LIN {X -326.728,Y -20.251,Z -40.000,A 0.015,B 0.000,C 180.000} C_DIS
LIN {X -326.353,Y -19.738,Z -40.000,A 0.015,B 0.000,C 180.000} C_DIS
LIN {X -324.173,Y -16.080,Z -40.000,A 0.015,B -0.000,C -180.000} C_DIS
LIN {X -324.033,Y -15.821,Z -40.000,A 0.015,B -0.000,C 180.000} C_DIS
LIN {X -323.375,Y -14.460,Z -40.000,A 0.015,B -0.000,C 180.000} C_DIS
LIN {X -323.235,Y -14.127,Z -40.000,A 0.015,B 0.000,C 180.000} C_DIS
LIN {X -321.515,Y -9.322,Z -40.000,A 0.015,B 0.000,C -180.000} C_DIS
LIN {X -321.341,Y -8.587,Z -40.000,A 0.015,B 0.000,C 180.000} C_DIS
LIN {X -320.684,Y -3.146,Z -40.000,A 0.015,B -0.000,C -180.000} C_DIS
LIN {X -320.667,Y -2.972,Z -40.000,A 0.015,B 0.000,C -180.000} C_DIS
LIN {X -320.518,Y -0.795,Z -40.000,A 0.015,B 0.000,C -180.000} C_DIS
LIN {X -320.520,Y -0.308,Z -40.000,A 0.015,B -0.000,C 180.000} C_DIS
LIN {X -320.740,Y 2.593,Z -40.000,A 0.015,B -0.000,C 180.000} C_DIS
LIN {X -320.791,Y 2.977,Z -40.000,A 0.015,B 0.000,C -180.000} C_DIS
LIN {X -321.349,Y 5.879,Z -40.000,A 0.015,B 0.000,C 180.000} C_DIS
LIN {X -321.416,Y 6.162,Z -40.000,A 0.015,B -0.000,C 180.000} C_DIS
LIN {X -321.819,Y 7.584,Z -40.000,A 0.015,B 0.000,C -180.000} C_DIS
LIN {X -321.946,Y 7.949,Z -40.000,A 0.015,B -0.000,C -180.000} C_DIS
LIN {X -324.346,Y 13.782,Z -40.000,A 0.015,B 0.000,C -180.000} C_DIS
LIN {X -324.544,Y 14.184,Z -40.000,A 0.015,B 0.000,C 180.000} C_DIS
LIN {X -342.684,Y 45.663,Z -40.000,A 0.015,B 0.000,C 180.000} C_DIS
LIN {X -342.906,Y 46.000,Z -40.000,A 0.015,B 0.000,C 180.000} C_DIS
LIN {X -344.864,Y 48.619,Z -40.000,A 0.015,B -0.000,C -180.000} C_DIS
LIN {X -344.919,Y 48.690,Z -40.000,A 0.015,B 0.000,C -180.000} C_DIS
LIN {X -347.449,Y 51.891,Z -40.000,A 0.015,B 0.000,C -180.000} C_DIS
LIN {X -347.826,Y 52.295,Z -40.000,A 0.015,B 0.000,C -180.000} C_DIS
LIN {X -350.266,Y 54.515,Z -40.000,A 0.015,B -0.000,C 180.000} C_DIS
LIN {X -350.603,Y 54.784,Z -40.000,A 0.015,B -0.000,C 180.000} C_DIS
LIN {X -352.993,Y 56.456,Z -40.000,A 0.015,B -0.000,C 180.000} C_DIS
LIN {X -353.258,Y 56.623,Z -40.000,A 0.015,B 0.000,C -180.000} C_DIS
LIN {X -354.709,Y 57.450,Z -40.000,A 0.015,B -0.000,C -180.000} C_DIS
LIN {X -355.032,Y 57.611,Z -40.000,A 0.015,B 0.000,C 180.000} C_DIS
LIN {X -360.836,Y 60.141,Z -40.000,A 0.015,B 0.000,C 180.000} C_DIS
LIN {X -361.547,Y 60.361,Z -40.000,A 0.015,B -0.000,C -180.000} C_DIS
LIN {X -365.901,Y 61.201,Z -40.000,A 0.015,B 0.000,C 180.000} C_DIS
LIN {X -366.162,Y 61.241,Z -40.000,A 0.015,B -0.000,C 180.000} C_DIS
LIN {X -368.338,Y 61.486,Z -40.000,A 0.015,B 0.000,C -180.000} C_DIS
LIN {X -368.781,Y 61.507,Z -40.000,A 0.015,B 0.000,C -180.000} C_DIS
LIN {X -373.497,Y 61.419,Z -40.000,A 0.015,B -0.000,C -180.000} C_DIS
LIN {X -374.399,Y 61.279,Z -40.000,A 0.015,B 0.000,C 180.000} C_DIS
LIN {X -383.592,Y 58.540,Z -40.000,A 0.015,B 0.000,C -180.000} C_DIS
LIN {X -383.923,Y 58.423,Z -40.000,A 0.015,B -0.000,C 180.000} C_DIS
LIN {X -384.920,Y 58.009,Z -40.000,A 0.015,B 0.000,C 180.000} C_DIS
LIN {X -385.722,Y 57.537,Z -40.000,A 0.015,B 0.000,C -180.000} C_DIS
LIN {X -393.652,Y 51.259,Z -40.000,A 0.015,B 0.000,C 180.000} C_DIS
LIN {X -394.115,Y 50.815,Z -40.000,A 0.015,B -0.000,C -180.000} C_DIS
LIN {X -395.224,Y 49.527,Z -40.000,A 0.015,B 0.000,C 180.000} C_DIS
LIN {X -395.515,Y 49.136,Z -40.000,A 0.015,B 0.000,C -180.000} C_DIS
LIN {X -397.824,Y 45.507,Z -40.000,A 0.015,B 0.000,C 180.000} C_DIS
LIN {X -397.891,Y 45.398,Z -40.000,A 0.015,B -0.000,C -180.000} C_DIS
LIN {X -401.772,Y 38.756,Z -40.000,A 0.015,B 0.000,C 180.000} C_DIS
LIN {X -401.996,Y 38.296,Z -40.000,A 0.015,B 0.000,C 180.000} C_DIS
LIN {X -402.542,Y 36.920,Z -40.000,A 0.015,B 0.000,C -180.000} C_DIS
LIN {X -402.687,Y 36.460,Z -40.000,A 0.015,B 0.000,C 180.000} C_DIS
LIN {X -403.779,Y 31.896,Z -40.000,A 0.015,B 0.000,C -180.000} C_DIS
LIN {X -403.787,Y 333.800,Z -40.000,A 0.015,B 0.000,C -180.000} C_DIS
LIN {X -403.730,Y 334.871,Z -40.000,A 0.015,B 0.000,C 180.000} C_DIS
LIN {X -403.533,Y 335.736,Z -40.000,A 0.015,B 0.000,C 180.000} C_DIS
LIN {X -403.418,Y 336.003,Z -40.000,A 0.015,B -0.000,C -180.000} C_DIS
LIN {X -403.034,Y 336.500,Z -39.830,A 0.015,B 0.000,C 180.000} C_DIS
LIN {X -402.624,Y 336.714,Z -39.365,A 0.015,B 0.000,C -180.000} C_DIS
LIN {X -402.458,Y 336.753,Z -38.730,A 0.015,B 0.000,C -180.000} C_DIS
$VEL.CP = 1.00000
LIN {X -402.458,Y 336.753,Z 11.000,A 0.015,B 0.000,C 180.000} C_DIS
$VEL.CP = 1.00000
LIN {X -176.907,Y 111.466,Z 11.000,A 0.015,B 0.000,C 180.000} C_DIS
$VEL.CP = 1.00000
LIN {X -176.907,Y 111.466,Z -28.231,A 0.015,B 0.000,C 180.000} C_DIS
$VEL.CP = 0.10000
LIN {X -176.826,Y 111.561,Z -28.780,A 0.015,B 0.000,C 180.000} C_DIS
LIN {X -176.608,Y 111.835,Z -29.221,A 0.015,B 0.000,C -180.000} C_DIS
LIN {X -176.404,Y 112.123,Z -29.421,A 0.015,B -0.000,C 180.000} C_DIS
LIN {X -176.196,Y 112.462,Z -29.500,A 0.015,B 0.000,C 180.000} C_DIS
LIN {X -176.625,Y 119.097,Z -29.746,A 0.015,B 0.000,C 180.000} C_DIS
LIN {X -182.895,Y 121.307,Z -29.992,A 0.015,B -0.000,C 180.000} C_DIS
LIN {X -187.390,Y 116.408,Z -30.238,A 0.015,B 0.000,C 180.000} C_DIS
LIN {X -184.650,Y 110.351,Z -30.484,A 0.015,B -0.000,C -180.000} C_DIS
LIN {X -178.003,Y 110.493,Z -30.730,A 0.015,B 0.000,C -180.000} C_DIS
LIN {X -175.523,Y 116.662,Z -30.975,A 0.015,B 0.000,C 180.000} C_DIS
LIN {X -180.223,Y 121.364,Z -31.221,A 0.015,B -0.000,C 180.000} C_DIS
LIN {X -186.394,Y 118.888,Z -31.467,A 0.015,B 0.000,C 180.000} C_DIS
LIN {X -186.539,Y 112.241,Z -31.713,A 0.015,B -0.000,C 180.000} C_DIS
LIN {X -180.483,Y 109.497,Z -31.959,A 0.015,B -0.000,C 180.000} C_DIS
LIN {X -175.582,Y 113.990,Z -32.205,A 0.015,B 0.000,C -180.000} C_DIS
LIN {X -177.789,Y 120.261,Z -32.451,A 0.015,B 0.000,C -180.000} C_DIS
LIN {X -184.423,Y 120.694,Z -32.697,A 0.015,B 0.000,C -180.000} C_DIS
LIN {X -187.426,Y 114.762,Z -32.943,A 0.015,B -0.000,C 180.000} C_DIS
LIN {X -183.150,Y 109.671,Z -33.189,A 0.015,B 0.000,C -180.000} C_DIS
LIN {X -176.789,Y 111.605,Z -33.434,A 0.015,B 0.000,C 180.000} C_DIS
LIN {X -176.070,Y 118.215,Z -33.680,A 0.015,B -0.000,C -180.000} C_DIS
LIN {X -181.867,Y 121.471,Z -33.926,A 0.015,B 0.000,C 180.000} C_DIS
LIN {X -187.137,Y 117.419,Z -34.172,A 0.015,B 0.000,C -180.000} C_DIS
LIN {X -185.480,Y 110.980,Z -34.418,A 0.015,B 0.000,C 180.000} C_DIS
LIN {X -178.907,Y 109.976,Z -34.664,A 0.015,B 0.000,C 180.000} C_DIS
LIN {X -175.404,Y 115.627,Z -34.910,A 0.015,B -0.000,C 180.000} C_DIS
LIN {X -179.225,Y 121.068,Z -35.156,A 0.015,B 0.000,C -180.000} C_DIS
LIN {X -185.729,Y 119.690,Z -35.402,A 0.015,B 0.000,C -180.000} C_DIS
LIN {X -187.016,Y 113.167,Z -35.648,A 0.015,B 0.000,C -180.000} C_DIS
LIN {X -181.522,Y 109.423,Z -35.893,A 0.015,B -0.000,C 180.000} C_DIS
LIN {X -175.921,Y 113.005,Z -36.139,A 0.015,B -0.000,C -180.000} C_DIS
LIN {X -177.016,Y 119.563,Z -36.385,A 0.015,B -0.000,C 180.000} C_DIS
LIN {X -183.478,Y 121.130,Z -36.631,A 0.015,B 0.000,C 180.000} C_DIS
LIN {X -187.456,Y 115.803,Z -36.877,A 0.015,B 0.000,C -180.000} C_DIS
LIN {X -184.119,Y 110.052,Z -37.123,A 0.015,B -0.000,C 180.000} C_DIS
LIN {X -177.520,Y 110.864,Z -37.369,A 0.015,B 0.000,C -180.000} C_DIS
LIN {X -175.675,Y 117.251,Z -37.615,A 0.015,B 0.000,C -180.000} C_DIS
LIN {X -180.825,Y 121.456,Z -37.861,A 0.015,B 0.000,C -180.000} C_DIS
LIN {X -186.715,Y 118.370,Z -38.107,A 0.015,B 0.000,C -180.000} C_DIS
LIN {X -186.189,Y 111.743,Z -38.352,A 0.015,B -0.000,C 180.000} C_DIS
LIN {X -179.887,Y 109.624,Z -38.598,A 0.015,B -0.000,C 180.000} C_DIS
LIN {X -175.464,Y 114.587,Z -38.844,A 0.015,B 0.000,C 180.000} C_DIS
LIN {X -178.292,Y 120.604,Z -39.090,A 0.015,B 0.000,C 180.000} C_DIS
LIN {X -184.937,Y 120.366,Z -39.336,A 0.015,B -0.000,C 180.000} C_DIS
LIN {X -187.326,Y 114.161,Z -39.582,A 0.015,B 0.000,C 180.000} C_DIS
LIN {X -182.558,Y 109.528,Z -39.828,A 0.015,B 0.000,C 180.000} C_DIS
LIN {X -176.424,Y 112.093,Z -40.074,A 0.015,B 0.000,C -180.000} C_DIS
LIN {X -176.376,Y 118.742,Z -40.320,A 0.015,B 0.000,C 180.000} C_DIS
LIN {X -182.471,Y 121.397,Z -40.566,A 0.015,B 0.000,C -180.000} C_DIS
LIN {X -187.306,Y 116.834,Z -40.811,A 0.015,B 0.000,C 180.000} C_DIS
LIN {X -185.008,Y 110.595,Z -41.057,A 0.015,B 0.000,C 180.000} C_DIS
LIN {X -178.368,Y 110.259,Z -41.303,A 0.015,B 0.000,C -180.000} C_DIS
LIN {X -175.452,Y 116.234,Z -41.549,A 0.015,B 0.000,C 180.000} C_DIS
LIN {X -179.802,Y 121.262,Z -41.795,A 0.015,B -0.000,C 180.000} C_DIS
LIN {X -186.134,Y 119.235,Z -42.041,A 0.015,B -0.000,C 180.000} C_DIS
LIN {X -186.757,Y 112.616,Z -42.287,A 0.015,B -0.000,C 180.000} C_DIS
LIN {X -180.913,Y 109.444,Z -42.533,A 0.015,B 0.000,C -180.000} C_DIS
LIN {X -175.702,Y 113.574,Z -42.779,A 0.015,B -0.000,C 180.000} C_DIS
LIN {X -177.453,Y 119.987,Z -43.025,A 0.015,B 0.000,C -180.000} C_DIS
LIN {X -184.040,Y 120.895,Z -43.270,A 0.015,B 0.000,C 180.000} C_DIS
LIN {X -187.461,Y 115.194,Z -43.516,A 0.015,B 0.000,C 180.000} C_DIS
LIN {X -183.560,Y 109.809,Z -43.762,A 0.015,B -0.000,C 180.000} C_DIS
LIN {X -177.077,Y 111.282,Z -44.008,A 0.015,B 0.000,C -180.000} C_DIS
LIN {X -175.886,Y 117.823,Z -44.254,A 0.015,B -0.000,C 180.000} C_DIS
LIN {X -181.434,Y 121.487,Z -44.500,A 0.015,B -0.000,C -180.000} C_DIS
LIN {X -214.171,Y 121.487,Z -44.500,A 0.015,B -0.000,C -180.000} C_DIS
CIRC {X -216.093,Y 120.378,Z -44.500,A 0.015,B -0.000,C 180.000},{X -216.095,Y 118.158,Z -44.500,A 0.015,B -0.000,C 180.000} C_DIS
LIN {X -214.870,Y 116.033,Z -44.500,A 0.015,B 0.000,C -180.000} C_DIS
CIRC {X -213.831,Y 114.992,Z -44.500,A 0.015,B 0.000,C -180.000},{X -212.410,Y 114.611,Z -44.500,A 0.015,B 0.000,C 180.000} C_DIS
LIN {X -181.088,Y 114.611,Z -44.500,A 0.015,B 0.000,C 180.000} C_DIS
CIRC {X -179.669,Y 114.991,Z -44.500,A 0.015,B 0.000,C 180.000},{X -178.630,Y 116.030,Z -44.500,A 0.015,B 0.000,C -180.000} C_DIS
LIN {X -177.403,Y 118.153,Z -44.500,A 0.015,B -0.000,C 180.000} C_DIS
CIRC {X -177.402,Y 120.375,Z -44.500,A 0.015,B 0.000,C -180.000},{X -179.327,Y 121.487,Z -44.500,A 0.015,B 0.000,C 180.000} C_DIS
LIN {X -181.434,Y 121.487,Z -44.500,A 0.015,B -0.000,C -180.000} C_DIS
CIRC {X -184.802,Y 122.507,Z -44.500,A 0.015,B 0.000,C -180.000},{X -187.038,Y 125.223,Z -44.500,A 0.015,B 0.000,C 180.000} C_DIS
CIRC {X -189.275,Y 127.940,Z -44.500,A 0.015,B 0.000,C 180.000},{X -192.643,Y 128.960,Z -44.500,A 0.015,B 0.000,C 180.000} C_DIS
LIN {X -214.895,Y 128.959,Z -44.500,A 0.015,B 0.000,C 180.000} C_DIS
CIRC {X -218.628,Y 129.066,Z -44.500,A 0.015,B -0.000,C -180.000},{X -222.348,Y 129.388,Z -44.500,A 0.015,B -0.000,C -180.000} C_DIS
CIRC {X -226.056,Y 129.807,Z -44.500,A 0.015,B 0.000,C 180.000},{X -229.767,Y 130.209,Z -44.500,A 0.015,B -0.000,C 180.000} C_DIS
CIRC {X -231.564,Y 129.293,Z -44.500,A 0.015,B -0.000,C -180.000},{X -231.455,Y 127.279,Z -44.500,A 0.015,B 0.000,C -180.000} C_DIS
CIRC {X -228.675,Y 123.312,Z -44.500,A 0.015,B 0.000,C -180.000},{X -226.050,Y 119.240,Z -44.500,A 0.015,B 0.000,C -180.000} C_DIS
CIRC {X -223.536,Y 115.099,Z -44.500,A 0.015,B 0.000,C -180.000},{X -221.085,Y 110.921,Z -44.500,A 0.015,B 0.000,C -180.000} C_DIS
CIRC {X -217.980,Y 107.812,Z -44.500,A 0.015,B 0.000,C 180.000},{X -213.736,Y 106.674,Z -44.500,A 0.015,B -0.000,C -180.000} C_DIS
LIN {X -179.775,Y 106.674,Z -44.500,A 0.015,B 0.000,C -180.000} C_DIS
CIRC {X -175.526,Y 107.812,Z -44.500,A 0.015,B 0.000,C -180.000},{X -172.415,Y 110.922,Z -44.500,A 0.015,B 0.000,C -180.000} C_DIS
CIRC {X -169.966,Y 115.093,Z -44.500,A 0.015,B 0.000,C 180.000},{X -167.463,Y 119.232,Z -44.500,A 0.015,B 0.000,C -180.000} C_DIS
CIRC {X -164.852,Y 123.304,Z -44.500,A 0.015,B 0.000,C 180.000},{X -162.086,Y 127.273,Z -44.500,A 0.015,B 0.000,C -180.000} C_DIS
CIRC {X -161.981,Y 129.289,Z -44.500,A 0.015,B 0.000,C -180.000},{X -163.780,Y 130.205,Z -44.500,A 0.015,B -0.000,C 180.000} C_DIS
CIRC {X -167.482,Y 129.805,Z -44.500,A 0.015,B 0.000,C 180.000},{X -171.182,Y 129.388,Z -44.500,A 0.015,B 0.000,C 180.000} C_DIS
CIRC {X -174.893,Y 129.067,Z -44.500,A 0.015,B 0.000,C 180.000},{X -178.617,Y 128.960,Z -44.500,A 0.015,B 0.000,C -180.000} C_DIS
LIN {X -192.643,Y 128.960,Z -44.500,A 0.015,B -0.000,C -180.000} C_DIS
CIRC {X -195.973,Y 129.957,Z -44.500,A 0.015,B 0.000,C -180.000},{X -198.206,Y 132.621,Z -44.500,A 0.015,B 0.000,C 180.000} C_DIS
CIRC {X -200.433,Y 135.294,Z -44.500,A 0.015,B -0.000,C 180.000},{X -203.768,Y 136.283,Z -44.500,A 0.015,B 0.000,C 180.000} C_DIS
LIN {X -214.895,Y 136.251,Z -44.500,A 0.015,B 0.000,C -180.000} C_DIS
CIRC {X -223.049,Y 136.543,Z -44.500,A 0.015,B 0.000,C -180.000},{X -231.161,Y 137.418,Z -44.500,A 0.015,B 0.000,C 180.000} C_DIS
CIRC {X -239.218,Y 138.678,Z -44.500,A 0.015,B 0.000,C 180.000},{X -247.242,Y 140.131,Z -44.500,A 0.015,B 0.000,C 180.000} C_DIS
CIRC {X -248.958,Y 139.347,Z -44.500,A 0.015,B -0.000,C -180.000},{X -248.776,Y 137.468,Z -44.500,A 0.015,B 0.000,C -180.000} C_DIS
CIRC {X -243.482,Y 131.173,Z -44.500,A 0.015,B -0.000,C -180.000},{X -238.409,Y 124.699,Z -44.500,A 0.015,B -0.000,C -180.000} C_DIS
CIRC {X -233.653,Y 117.984,Z -44.500,A 0.015,B -0.000,C -180.000},{X -229.325,Y 110.986,Z -44.500,A 0.015,B 0.000,C 180.000} C_DIS
CIRC {X -228.301,Y 109.143,Z -44.500,A 0.015,B 0.000,C 180.000},{X -227.335,Y 107.269,Z -44.500,A 0.015,B 0.000,C 180.000} C_DIS
CIRC {X -226.368,Y 105.394,Z -44.500,A 0.015,B 0.000,C -180.000},{X -225.344,Y 103.551,Z -44.500,A 0.015,B 0.000,C -180.000} C_DIS
CIRC {X -222.239,Y 100.442,Z -44.500,A 0.015,B 0.000,C -180.000},{X -217.995,Y 99.304,Z -44.500,A 0.015,B 0.000,C -180.000} C_DIS
LIN {X -175.522,Y 99.304,Z -44.500,A 0.015,B 0.000,C -180.000} C_DIS
CIRC {X -171.273,Y 100.442,Z -44.500,A 0.015,B -0.000,C 180.000},{X -168.162,Y 103.552,Z -44.500,A 0.015,B 0.000,C -180.000} C_DIS
CIRC {X -167.074,Y 105.503,Z -44.500,A 0.015,B -0.000,C 180.000},{X -166.049,Y 107.487,Z -44.500,A 0.015,B -0.000,C -180.000} C_DIS
CIRC {X -165.023,Y 109.471,Z -44.500,A 0.015,B 0.000,C -180.000},{X -163.936,Y 111.422,Z -44.500,A 0.015,B -0.000,C -180.000} C_DIS
CIRC {X -159.658,Y 118.305,Z -44.500,A 0.015,B -0.000,C -180.000},{X -154.949,Y 124.900,Z -44.500,A 0.015,B -0.000,C -180.000} C_DIS
CIRC {X -149.935,Y 131.262,Z -44.500,A 0.015,B 0.000,C 180.000},{X -144.727,Y 137.467,Z -44.500,A 0.015,B 0.000,C -180.000} C_DIS
CIRC {X -144.548,Y 139.348,Z -44.500,A 0.015,B 0.000,C 180.000},{X -146.267,Y 140.131,Z -44.500,A 0.015,B 0.000,C -180.000} C_DIS
CIRC {X -163.300,Y 137.597,Z -44.500,A 0.015,B 0.000,C -180.000},{X -180.488,Y 136.550,Z -44.500,A 0.015,B 0.000,C -180.000} C_DIS
LIN {X -203.768,Y 136.283,Z -44.500,A 0.015,B 0.000,C -180.000} C_DIS
CIRC {X -206.836,Y 137.199,Z -44.500,A 0.015,B 0.000,C 180.000},{X -208.871,Y 139.672,Z -44.500,A 0.015,B 0.000,C -180.000} C_DIS
CIRC {X -210.910,Y 142.136,Z -44.500,A 0.015,B 0.000,C 180.000},{X -213.973,Y 143.061,Z -44.500,A 0.015,B 0.000,C -180.000} C_DIS
LIN {X -214.895,Y 143.061,Z -44.500,A 0.015,B 0.000,C 180.000} C_DIS
CIRC {X -230.275,Y 143.896,Z -44.500,A 0.015,B 0.000,C 180.000},{X -245.474,Y 146.392,Z -44.500,A 0.015,B 0.000,C 180.000} C_DIS
CIRC {X -260.344,Y 150.380,Z -44.500,A 0.015,B 0.000,C -180.000},{X -274.796,Y 155.687,Z -44.500,A 0.015,B 0.000,C 180.000} C_DIS
CIRC {X -276.352,Y 155.160,Z -44.500,A 0.015,B 0.000,C -180.000},{X -276.023,Y 153.551,Z -44.500,A 0.015,B 0.000,C 180.000} C_DIS
CIRC {X -267.113,Y 146.298,Z -44.500,A 0.015,B 0.000,C -180.000},{X -258.772,Y 138.398,Z -44.500,A 0.015,B -0.000,C 180.000} C_DIS
CIRC {X -250.999,Y 129.940,Z -44.500,A 0.015,B -0.000,C 180.000},{X -243.781,Y 121.005,Z -44.500,A 0.015,B 0.000,C 180.000} C_DIS
CIRC {X -241.444,Y 117.780,Z -44.500,A 0.015,B 0.000,C -180.000},{X -239.241,Y 114.462,Z -44.500,A 0.015,B -0.000,C 180.000} C_DIS
CIRC {X -237.143,Y 111.077,Z -44.500,A 0.015,B 0.000,C 180.000},{X -235.118,Y 107.648,Z -44.500,A 0.015,B -0.000,C 180.000} C_DIS
CIRC {X -233.616,Y 104.944,Z -44.500,A 0.015,B 0.000,C -180.000},{X -232.199,Y 102.195,Z -44.500,A 0.015,B 0.000,C 180.000} C_DIS
CIRC {X -230.782,Y 99.445,Z -44.500,A 0.015,B 0.000,C 180.000},{X -229.279,Y 96.742,Z -44.500,A 0.015,B 0.000,C 180.000} C_DIS
CIRC {X -226.174,Y 93.633,Z -44.500,A 0.015,B 0.000,C 180.000},{X -221.930,Y 92.495,Z -44.500,A 0.015,B 0.000,C -180.000} C_DIS
LIN {X -171.593,Y 92.495,Z -44.500,A 0.015,B 0.000,C 180.000} C_DIS
CIRC {X -167.344,Y 93.633,Z -44.500,A 0.015,B 0.000,C 180.000},{X -164.232,Y 96.743,Z -44.500,A 0.015,B 0.000,C -180.000} C_DIS
CIRC {X -162.667,Y 99.552,Z -44.500,A 0.015,B 0.000,C -180.000},{X -161.189,Y 102.409,Z -44.500,A 0.015,B 0.000,C -180.000} C_DIS
CIRC {X -159.712,Y 105.266,Z -44.500,A 0.015,B -0.000,C 180.000},{X -158.147,Y 108.076,Z -44.500,A 0.015,B 0.000,C -180.000} C_DIS
CIRC {X -149.761,Y 120.950,Z -44.500,A 0.015,B 0.000,C -180.000},{X -140.052,Y 132.859,Z -44.500,A 0.015,B -0.000,C -180.000} C_DIS
CIRC {X -129.216,Y 143.744,Z -44.500,A 0.015,B 0.000,C -180.000},{X -117.430,Y 153.592,Z -44.500,A 0.015,B 0.000,C 180.000} C_DIS
CIRC {X -117.109,Y 155.202,Z -44.500,A 0.015,B 0.000,C 180.000},{X -118.667,Y 155.719,Z -44.500,A 0.015,B -0.000,C 180.000} C_DIS
CIRC {X -129.206,Y 151.681,Z -44.500,A 0.015,B -0.000,C 180.000},{X -140.015,Y 148.432,Z -44.500,A 0.015,B 0.000,C 180.000} C_DIS
CIRC {X -151.019,Y 145.931,Z -44.500,A 0.015,B 0.000,C -180.000},{X -162.157,Y 144.126,Z -44.500,A 0.015,B -0.000,C -180.000} C_DIS
CIRC {X -170.370,Y 143.327,Z -44.500,A 0.015,B -0.000,C -180.000},{X -178.617,Y 143.061,Z -44.500,A 0.015,B 0.000,C -180.000} C_DIS
LIN {X -213.973,Y 143.061,Z -44.500,A 0.015,B 0.000,C 180.000} C_DIS
CIRC {X -217.010,Y 143.987,Z -44.500,A 0.015,B -0.000,C -180.000},{X -219.013,Y 146.452,Z -44.500,A 0.015,B -0.000,C 180.000} C_DIS
CIRC {X -220.965,Y 148.937,Z -44.500,A 0.015,B 0.000,C -180.000},{X -223.938,Y 150.007,Z -44.500,A 0.015,B 0.000,C 180.000} C_DIS
CIRC {X -237.131,Y 151.527,Z -44.500,A 0.015,B -0.000,C 180.000},{X -250.115,Y 154.318,Z -44.500,A 0.015,B 0.000,C -180.000} C_DIS
CIRC {X -267.037,Y 159.791,Z -44.500,A 0.015,B 0.000,C 180.000},{X -283.292,Y 167.008,Z -44.500,A 0.015,B 0.000,C -180.000} C_DIS
CIRC {X -285.560,Y 166.917,Z -44.500,A 0.015,B -0.000,C 180.000},{X -286.669,Y 164.936,Z -44.500,A 0.015,B 0.000,C -180.000} C_DIS
LIN {X -286.669,Y 156.530,Z -44.500,A 0.015,B 0.000,C 180.000} C_DIS
CIRC {X -285.894,Y 153.375,Z -44.500,A 0.015,B 0.000,C 180.000},{X -283.747,Y 150.938,Z -44.500,A 0.015,B 0.000,C 180.000} C_DIS
CIRC {X -274.065,Y 143.550,Z -44.500,A 0.015,B 0.000,C 180.000},{X -265.073,Y 135.336,Z -44.500,A 0.015,B -0.000,C 180.000} C_DIS
CIRC {X -256.759,Y 126.443,Z -44.500,A 0.015,B 0.000,C 180.000},{X -249.083,Y 116.994,Z -44.500,A 0.015,B 0.000,C 180.000} C_DIS
CIRC {X -244.724,Y 110.826,Z -44.500,A 0.015,B 0.000,C 180.000},{X -240.774,Y 104.389,Z -44.500,A 0.015,B 0.000,C 180.000} C_DIS
CIRC {X -238.805,Y 100.845,Z -44.500,A 0.015,B 0.000,C 180.000},{X -236.947,Y 97.241,Z -44.500,A 0.015,B -0.000,C 180.000} C_DIS
CIRC {X -235.090,Y 93.638,Z -44.500,A 0.015,B 0.000,C -180.000},{X -233.121,Y 90.094,Z -44.500,A 0.015,B -0.000,C -180.000} C_DIS
CIRC {X -230.016,Y 86.985,Z -44.500,A 0.015,B 0.000,C 180.000},{X -225.772,Y 85.847,Z -44.500,A 0.015,B -0.000,C 180.000} C_DIS
LIN {X -167.757,Y 85.847,Z -44.500,A 0.015,B 0.000,C 180.000} C_DIS
CIRC {X -163.508,Y 86.985,Z -44.500,A 0.015,B -0.000,C -180.000},{X -160.396,Y 90.095,Z -44.500,A 0.015,B 0.000,C -180.000} C_DIS
CIRC {X -158.363,Y 93.743,Z -44.500,A 0.015,B 0.000,C 180.000},{X -156.445,Y 97.452,Z -44.500,A 0.015,B 0.000,C 180.000} C_DIS
CIRC {X -154.528,Y 101.162,Z -44.500,A 0.015,B 0.000,C 180.000},{X -152.495,Y 104.810,Z -44.500,A 0.015,B -0.000,C -180.000} C_DIS
CIRC {X -143.792,Y 118.058,Z -44.500,A 0.015,B -0.000,C 180.000},{X -133.633,Y 130.226,Z -44.500,A 0.015,B 0.000,C -180.000} C_DIS
CIRC {X -122.219,Y 141.219,Z -44.500,A 0.015,B 0.000,C -180.000},{X -109.738,Y 150.983,Z -44.500,A 0.015,B 0.000,C -180.000} C_DIS
CIRC {X -107.610,Y 153.416,Z -44.500,A 0.015,B 0.000,C 180.000},{X -106.843,Y 156.556,Z -44.500,A 0.015,B 0.000,C 180.000} C_DIS
LIN {X -106.843,Y 164.935,Z -44.500,A 0.015,B 0.000,C 180.000} C_DIS
CIRC {X -107.952,Y 166.917,Z -44.500,A 0.015,B 0.000,C 180.000},{X -110.221,Y 167.007,Z -44.500,A 0.015,B 0.000,C -180.000} C_DIS
CIRC {X -116.135,Y 164.079,Z -44.500,A 0.015,B 0.000,C 180.000},{X -122.111,Y 161.278,Z -44.500,A 0.015,B 0.000,C 180.000} C_DIS
CIRC {X -128.194,Y 158.712,Z -44.500,A 0.015,B 0.000,C -180.000},{X -134.413,Y 156.498,Z -44.500,A 0.015,B 0.000,C 180.000} C_DIS
CIRC {X -154.153,Y 151.711,Z -44.500,A 0.015,B -0.000,C -180.000},{X -174.388,Y 149.944,Z -44.500,A 0.015,B 0.000,C 180.000} C_DIS
LIN {X -214.895,Y 149.708,Z -44.500,A 0.015,B 0.000,C -180.000} C_DIS
CIRC {X -219.419,Y 149.783,Z -44.500,A 0.015,B 0.000,C -180.000},{X -223.938,Y 150.007,Z -44.500,A 0.015,B 0.000,C -180.000} C_DIS
CIRC {X -227.574,Y 151.391,Z -44.500,A 0.015,B 0.000,C 180.000},{X -229.811,Y 154.574,Z -44.500,A 0.015,B 0.000,C 180.000} C_DIS
CIRC {X -231.967,Y 157.783,Z -44.500,A 0.015,B 0.000,C -180.000},{X -235.486,Y 159.385,Z -44.500,A 0.015,B -0.000,C 180.000} C_DIS
CIRC {X -264.728,Y 167.211,Z -44.500,A 0.015,B 0.000,C -180.000},{X -291.539,Y 181.267,Z -44.500,A 0.015,B 0.000,C -180.000} C_DIS
CIRC {X -293.684,Y 181.380,Z -44.500,A 0.015,B 0.000,C 180.000},{X -294.790,Y 179.539,Z -44.500,A 0.015,B 0.000,C 180.000} C_DIS
LIN {X -294.790,Y 153.838,Z -44.500,A 0.015,B 0.000,C 180.000} C_DIS
CIRC {X -293.674,Y 149.301,Z -44.500,A 0.015,B 0.000,C 180.000},{X -290.583,Y 145.798,Z -44.500,A 0.015,B -0.000,C 180.000} C_DIS
CIRC {X -282.137,Y 139.589,Z -44.500,A 0.015,B 0.000,C 180.000},{X -274.042,Y 132.930,Z -44.500,A 0.015,B 0.000,C -180.000} C_DIS
CIRC {X -266.491,Y 125.644,Z -44.500,A 0.015,B 0.000,C -180.000},{X -259.735,Y 117.616,Z -44.500,A 0.015,B 0.000,C 180.000} C_DIS
CIRC {X -256.589,Y 113.410,Z -44.500,A 0.015,B -0.000,C 180.000},{X -253.487,Y 109.171,Z -44.500,A 0.015,B 0.000,C -180.000} C_DIS
CIRC {X -250.519,Y 104.836,Z -44.500,A 0.015,B 0.000,C -180.000},{X -247.778,Y 100.352,Z -44.500,A 0.015,B 0.000,C -180.000} C_DIS
CIRC {X -245.228,Y 95.790,Z -44.500,A 0.015,B 0.000,C 180.000},{X -242.796,Y 91.163,Z -44.500,A 0.015,B 0.000,C 180.000} C_DIS
CIRC {X -240.365,Y 86.536,Z -44.500,A 0.015,B -0.000,C 180.000},{X -237.814,Y 81.973,Z -44.500,A 0.015,B 0.000,C 180.000} C_DIS
CIRC {X -234.709,Y 78.865,Z -44.500,A 0.015,B 0.000,C -180.000},{X -230.465,Y 77.726,Z -44.500,A 0.015,B 0.000,C -180.000} C_DIS
LIN {X -163.071,Y 77.726,Z -44.500,A 0.015,B 0.000,C 180.000} C_DIS
CIRC {X -158.821,Y 78.865,Z -44.500,A 0.015,B 0.000,C -180.000},{X -155.710,Y 81.974,Z -44.500,A 0.015,B -0.000,C 180.000} C_DIS
CIRC {X -153.093,Y 86.637,Z -44.500,A 0.015,B 0.000,C 180.000},{X -150.596,Y 91.366,Z -44.500,A 0.015,B 0.000,C -180.000} C_DIS
CIRC {X -148.099,Y 96.094,Z -44.500,A 0.015,B 0.000,C -180.000},{X -145.482,Y 100.757,Z -44.500,A 0.015,B 0.000,C 180.000} C_DIS
CIRC {X -136.887,Y 113.783,Z -44.500,A 0.015,B 0.000,C 180.000},{X -126.813,Y 125.701,Z -44.500,A 0.015,B 0.000,C 180.000} C_DIS
CIRC {X -115.449,Y 136.392,Z -44.500,A 0.015,B 0.000,C -180.000},{X -102.981,Y 145.772,Z -44.500,A 0.015,B -0.000,C 180.000} C_DIS
CIRC {X -99.854,Y 149.227,Z -44.500,A 0.015,B 0.000,C -180.000},{X -98.722,Y 153.749,Z -44.500,A 0.015,B 0.000,C -180.000} C_DIS
LIN {X -98.723,Y 179.538,Z -44.500,A 0.015,B 0.000,C -180.000} C_DIS
CIRC {X -99.829,Y 181.379,Z -44.500,A 0.015,B -0.000,C -180.000},{X -101.974,Y 181.266,Z -44.500,A 0.015,B 0.000,C -180.000} C_DIS
CIRC {X -116.357,Y 172.865,Z -44.500,A 0.015,B 0.000,C 180.000},{X -131.706,Y 166.399,Z -44.500,A 0.015,B -0.000,C -180.000} C_DIS
CIRC {X -147.689,Y 161.757,Z -44.500,A 0.015,B 0.000,C -180.000},{X -164.061,Y 158.771,Z -44.500,A 0.015,B 0.000,C -180.000} C_DIS
CIRC {X -171.324,Y 158.065,Z -44.500,A 0.015,B 0.000,C 180.000},{X -178.617,Y 157.829,Z -44.500,A 0.015,B -0.000,C -180.000} C_DIS
LIN {X -214.895,Y 157.829,Z -44.500,A 0.015,B 0.000,C -180.000} C_DIS
CIRC {X -225.220,Y 158.218,Z -44.500,A 0.015,B -0.000,C -180.000},{X -235.486,Y 159.385,Z -44.500,A 0.015,B 0.000,C -180.000} C_DIS
CIRC {X -238.870,Y 161.018,Z -44.500,A 0.015,B 0.000,C -180.000},{X -240.750,Y 164.273,Z -44.500,A 0.015,B -0.000,C 180.000} C_DIS
CIRC {X -242.541,Y 167.547,Z -44.500,A 0.015,B 0.000,C -180.000},{X -245.782,Y 169.399,Z -44.500,A 0.015,B 0.000,C 180.000} C_DIS
CIRC {X -260.443,Y 173.863,Z -44.500,A 0.015,B 0.000,C 180.000},{X -274.560,Y 179.825,Z -44.500,A 0.015,B 0.000,C -180.000} C_DIS
CIRC {X -281.181,Y 183.420,Z -44.500,A 0.015,B 0.000,C -180.000},{X -287.445,Y 187.607,Z -44.500,A 0.015,B 0.000,C 180.000} C_DIS
CIRC {X -293.465,Y 192.125,Z -44.500,A 0.015,B 0.000,C 180.000},{X -299.406,Y 196.745,Z -44.500,A 0.015,B 0.000,C 180.000} C_DIS
CIRC {X -301.473,Y 196.972,Z -44.500,A 0.015,B 0.000,C -180.000},{X -302.577,Y 195.211,Z -44.500,A 0.015,B 0.000,C -180.000} C_DIS
LIN {X -302.576,Y 149.343,Z -44.500,A 0.015,B 0.000,C -180.000} C_DIS
CIRC {X -301.480,Y 145.018,Z -44.500,A 0.015,B 0.000,C 180.000},{X -298.458,Y 141.736,Z -44.500,A 0.015,B 0.000,C 180.000} C_DIS
CIRC {X -293.362,Y 138.324,Z -44.500,A 0.015,B 0.000,C -180.000},{X -288.344,Y 134.797,Z -44.500,A 0.015,B 0.000,C 180.000} C_DIS
CIRC {X -283.471,Y 131.069,Z -44.500,A 0.015,B 0.000,C -180.000},{X -278.825,Y 127.062,Z -44.500,A 0.015,B 0.000,C -180.000} C_DIS
CIRC {X -271.868,Y 120.152,Z -44.500,A 0.015,B 0.000,C 180.000},{X -265.498,Y 112.698,Z -44.500,A 0.015,B -0.000,C -180.000} C_DIS
CIRC {X -259.720,Y 104.778,Z -44.500,A 0.015,B 0.000,C -180.000},{X -254.524,Y 96.465,Z -44.500,A 0.015,B -0.000,C 180.000} C_DIS
LIN {X -242.314,Y 74.187,Z -44.500,A 0.015,B -0.000,C 180.000} C_DIS
CIRC {X -239.209,Y 71.078,Z -44.500,A 0.015,B 0.000,C 180.000},{X -234.965,Y 69.940,Z -44.500,A 0.015,B 0.000,C 180.000} C_DIS
LIN {X -158.577,Y 69.940,Z -44.500,A 0.015,B -0.000,C 180.000} C_DIS
CIRC {X -154.328,Y 71.078,Z -44.500,A 0.015,B 0.000,C -180.000},{X -151.217,Y 74.188,Z -44.500,A 0.015,B 0.000,C -180.000} C_DIS
LIN {X -138.741,Y 96.861,Z -44.500,A 0.015,B 0.000,C 180.000} C_DIS
CIRC {X -132.579,Y 106.475,Z -44.500,A 0.015,B 0.000,C -180.000},{X -125.560,Y 115.482,Z -44.500,A 0.015,B 0.000,C 180.000} C_DIS
CIRC {X -117.826,Y 123.876,Z -44.500,A 0.015,B -0.000,C -180.000},{X -109.498,Y 131.681,Z -44.500,A 0.015,B 0.000,C 180.000} C_DIS
CIRC {X -106.071,Y 134.441,Z -44.500,A 0.015,B 0.000,C 180.000},{X -102.443,Y 136.928,Z -44.500,A 0.015,B -0.000,C -180.000} C_DIS
CIRC {X -98.737,Y 139.292,Z -44.500,A 0.015,B -0.000,C 180.000},{X -95.054,Y 141.692,Z -44.500,A 0.015,B 0.000,C 180.000} C_DIS
CIRC {X -92.031,Y 144.997,Z -44.500,A 0.015,B 0.000,C -180.000},{X -90.936,Y 149.339,Z -44.500,A 0.015,B 0.000,C 180.000} C_DIS
LIN {X -90.937,Y 195.209,Z -44.500,A 0.015,B 0.000,C 180.000} C_DIS
CIRC {X -92.042,Y 196.970,Z -44.500,A 0.015,B 0.000,C 180.000},{X -94.108,Y 196.743,Z -44.500,A 0.015,B 0.000,C -180.000} C_DIS
CIRC {X -101.145,Y 191.386,Z -44.500,A 0.015,B -0.000,C 180.000},{X -108.380,Y 186.298,Z -44.500,A 0.015,B 0.000,C 180.000} C_DIS
CIRC {X -115.899,Y 181.631,Z -44.500,A 0.015,B 0.000,C -180.000},{X -123.755,Y 177.556,Z -44.500,A 0.015,B 0.000,C 180.000} C_DIS
CIRC {X -133.687,Y 173.478,Z -44.500,A 0.015,B 0.000,C 180.000},{X -143.979,Y 170.417,Z -44.500,A 0.015,B 0.000,C -180.000} C_DIS
CIRC {X -154.468,Y 168.166,Z -44.500,A 0.015,B 0.000,C -180.000},{X -165.065,Y 166.492,Z -44.500,A 0.015,B 0.000,C -180.000} C_DIS
CIRC {X -171.827,Y 165.835,Z -44.500,A 0.015,B 0.000,C 180.000},{X -178.617,Y 165.615,Z -44.500,A 0.015,B 0.000,C 180.000} C_DIS
LIN {X -214.895,Y 165.615,Z -44.500,A 0.015,B 0.000,C 180.000} C_DIS
CIRC {X -230.327,Y 166.549,Z -44.500,A 0.015,B -0.000,C 180.000},{X -245.533,Y 169.338,Z -44.500,A 0.015,B 0.000,C 180.000} C_DIS
LIN {X -245.782,Y 169.399,Z -44.500,A 0.015,B 0.000,C 180.000} C_DIS
CIRC {X -248.841,Y 171.234,Z -44.500,A 0.015,B -0.000,C 180.000},{X -250.352,Y 174.465,Z -44.500,A 0.015,B -0.000,C 180.000} C_DIS
CIRC {X -251.788,Y 177.707,Z -44.500,A 0.015,B -0.000,C 180.000},{X -254.711,Y 179.713,Z -44.500,A 0.015,B -0.000,C 180.000} C_DIS
CIRC {X -260.134,Y 181.685,Z -44.500,A 0.015,B -0.000,C -180.000},{X -265.460,Y 183.905,Z -44.500,A 0.015,B 0.000,C 180.000} C_DIS
CIRC {X -287.951,Y 196.939,Z -44.500,A 0.015,B 0.000,C -180.000},{X -307.158,Y 214.454,Z -44.500,A 0.015,B 0.000,C -180.000} C_DIS
CIRC {X -309.038,Y 214.918,Z -44.500,A 0.015,B 0.000,C -180.000},{X -310.138,Y 213.325,Z -44.500,A 0.015,B -0.000,C 180.000} C_DIS
LIN {X -310.136,Y 144.758,Z -44.500,A 0.015,B 0.000,C 180.000} C_DIS
CIRC {X -309.041,Y 140.616,Z -44.500,A 0.015,B -0.000,C 180.000},{X -306.042,Y 137.557,Z -44.500,A 0.015,B 0.000,C -180.000} C_DIS
CIRC {X -295.237,Y 130.344,Z -44.500,A 0.015,B 0.000,C 180.000},{X -285.238,Y 122.050,Z -44.500,A 0.015,B 0.000,C 180.000} C_DIS
CIRC {X -276.089,Y 112.833,Z -44.500,A 0.015,B -0.000,C 180.000},{X -267.799,Y 102.837,Z -44.500,A 0.015,B -0.000,C 180.000} C_DIS
CIRC {X -264.279,Y 97.868,Z -44.500,A 0.015,B 0.000,C -180.000},{X -261.076,Y 92.690,Z -44.500,A 0.015,B -0.000,C -180.000} C_DIS
LIN {X -246.683,Y 66.626,Z -44.500,A 0.015,B 0.000,C 180.000} C_DIS
CIRC {X -243.578,Y 63.518,Z -44.500,A 0.015,B -0.000,C -180.000},{X -239.334,Y 62.379,Z -44.500,A 0.015,B 0.000,C -180.000} C_DIS
LIN {X -154.214,Y 62.379,Z -44.500,A 0.015,B 0.000,C -180.000} C_DIS
CIRC {X -149.965,Y 63.518,Z -44.500,A 0.015,B 0.000,C -180.000},{X -146.853,Y 66.627,Z -44.500,A 0.015,B 0.000,C -180.000} C_DIS
LIN {X -132.194,Y 93.078,Z -44.500,A 0.015,B -0.000,C 180.000} C_DIS
CIRC {X -123.292,Y 106.288,Z -44.500,A 0.015,B -0.000,C 180.000},{X -112.657,Y 118.148,Z -44.500,A 0.015,B 0.000,C 180.000} C_DIS
CIRC {X -100.621,Y 128.565,Z -44.500,A 0.015,B 0.000,C -180.000},{X -87.470,Y 137.535,Z -44.500,A 0.015,B 0.000,C -180.000} C_DIS
CIRC {X -84.470,Y 140.615,Z -44.500,A 0.015,B -0.000,C 180.000},{X -83.375,Y 144.774,Z -44.500,A 0.015,B 0.000,C 180.000} C_DIS
LIN {X -83.377,Y 213.321,Z -44.500,A 0.015,B -0.000,C 180.000} C_DIS
CIRC {X -84.477,Y 214.914,Z -44.500,A 0.015,B 0.000,C -180.000},{X -86.357,Y 214.450,Z -44.500,A 0.015,B 0.000,C 180.000} C_DIS
CIRC {X -103.087,Y 198.936,Z -44.500,A 0.015,B 0.000,C 180.000},{X -122.532,Y 187.000,Z -44.500,A 0.015,B -0.000,C -180.000} C_DIS
CIRC {X -143.760,Y 178.737,Z -44.500,A 0.015,B 0.000,C -180.000},{X -166.039,Y 173.990,Z -44.500,A 0.015,B 0.000,C 180.000} C_DIS
CIRC {X -172.315,Y 173.380,Z -44.500,A 0.015,B -0.000,C 180.000},{X -178.617,Y 173.176,Z -44.500,A 0.015,B 0.000,C 180.000} C_DIS
LIN {X -214.895,Y 173.176,Z -44.500,A 0.015,B 0.000,C 180.000} C_DIS
CIRC {X -235.070,Y 174.821,Z -44.500,A 0.015,B -0.000,C -180.000},{X -254.711,Y 179.713,Z -44.500,A 0.015,B -0.000,C 180.000} C_DIS
CIRC {X -257.492,Y 181.715,Z -44.500,A 0.015,B 0.000,C 180.000},{X -258.667,Y 184.934,Z -44.500,A 0.015,B -0.000,C -180.000} C_DIS
CIRC {X -259.761,Y 188.157,Z -44.500,A 0.015,B 0.000,C -180.000},{X -262.381,Y 190.329,Z -44.500,A 0.015,B 0.000,C -180.000} C_DIS
CIRC {X -291.818,Y 209.027,Z -44.500,A 0.015,B 0.000,C 180.000},{X -314.459,Y 235.551,Z -44.500,A 0.015,B -0.000,C -180.000} C_DIS
CIRC {X -316.156,Y 236.207,Z -44.500,A 0.015,B 0.000,C -180.000},{X -317.252,Y 234.755,Z -44.500,A 0.015,B 0.000,C 180.000} C_DIS
LIN {X -317.250,Y 140.220,Z -44.500,A 0.015,B -0.000,C -180.000} C_DIS
CIRC {X -316.155,Y 136.259,Z -44.500,A 0.015,B 0.000,C -180.000},{X -313.181,Y 133.423,Z -44.500,A 0.015,B -0.000,C 180.000} C_DIS
CIRC {X -301.847,Y 126.435,Z -44.500,A 0.015,B 0.000,C -180.000},{X -291.439,Y 118.132,Z -44.500,A 0.015,B 0.000,C -180.000} C_DIS
CIRC {X -281.992,Y 108.764,Z -44.500,A 0.015,B 0.000,C 180.000},{X -273.472,Y 98.545,Z -44.500,A 0.015,B -0.000,C 180.000} C_DIS
CIRC {X -270.209,Y 93.939,Z -44.500,A 0.015,B -0.000,C -180.000},{X -267.239,Y 89.138,Z -44.500,A 0.015,B 0.000,C -180.000} C_DIS
LIN {X -250.775,Y 59.479,Z -44.500,A 0.015,B -0.000,C 180.000} C_DIS
CIRC {X -247.694,Y 56.395,Z -44.500,A 0.015,B 0.000,C 180.000},{X -243.484,Y 55.266,Z -44.500,A 0.015,B 0.000,C 180.000} C_DIS
LIN {X -150.044,Y 55.266,Z -44.500,A 0.015,B -0.000,C 180.000} C_DIS
CIRC {X -145.851,Y 56.389,Z -44.500,A 0.015,B 0.000,C 180.000},{X -142.781,Y 59.457,Z -44.500,A 0.015,B 0.000,C -180.000} C_DIS
LIN {X -126.035,Y 89.519,Z -44.500,A 0.015,B -0.000,C 180.000} C_DIS
CIRC {X -117.034,Y 102.790,Z -44.500,A 0.015,B 0.000,C -180.000},{X -106.222,Y 114.633,Z -44.500,A 0.015,B -0.000,C -180.000} C_DIS
CIRC {X -93.894,Y 124.877,Z -44.500,A 0.015,B 0.000,C 180.000},{X -80.332,Y 133.421,Z -44.500,A 0.015,B 0.000,C 180.000} C_DIS
CIRC {X -77.356,Y 136.279,Z -44.500,A 0.015,B 0.000,C 180.000},{X -76.261,Y 140.257,Z -44.500,A 0.015,B 0.000,C -180.000} C_DIS
LIN {X -76.264,Y 234.747,Z -44.500,A 0.015,B 0.000,C -180.000} C_DIS
CIRC {X -77.360,Y 236.200,Z -44.500,A 0.015,B 0.000,C -180.000},{X -79.057,Y 235.544,Z -44.500,A 0.015,B 0.000,C 180.000} C_DIS
CIRC {X -91.630,Y 218.902,Z -44.500,A 0.015,B 0.000,C -180.000},{X -107.020,Y 204.824,Z -44.500,A 0.015,B 0.000,C 180.000} C_DIS
CIRC {X -124.620,Y 193.657,Z -44.500,A 0.015,B -0.000,C -180.000},{X -143.840,Y 185.591,Z -44.500,A 0.015,B 0.000,C 180.000} C_DIS
CIRC {X -161.281,Y 181.450,Z -44.500,A 0.015,B -0.000,C 180.000},{X -179.160,Y 180.151,Z -44.500,A 0.015,B 0.000,C -180.000} C_DIS
LIN {X -214.895,Y 180.290,Z -44.500,A 0.015,B 0.000,C 180.000} C_DIS
CIRC {X -239.163,Y 182.827,Z -44.500,A 0.015,B 0.000,C -180.000},{X -262.381,Y 190.329,Z -44.500,A 0.015,B 0.000,C -180.000} C_DIS
CIRC {X -264.753,Y 192.387,Z -44.500,A 0.015,B 0.000,C -180.000},{X -265.561,Y 195.420,Z -44.500,A 0.015,B 0.000,C -180.000} C_DIS
CIRC {X -266.299,Y 198.451,Z -44.500,A 0.015,B 0.000,C 180.000},{X -268.518,Y 200.644,Z -44.500,A 0.015,B 0.000,C 180.000} C_DIS
CIRC {X -298.382,Y 224.614,Z -44.500,A 0.015,B 0.000,C -180.000},{X -318.342,Y 257.296,Z -44.500,A 0.015,B 0.000,C -180.000} C_DIS
CIRC {X -321.512,Y 259.045,Z -44.500,A 0.015,B 0.000,C 180.000},{X -323.822,Y 256.256,Z -44.500,A 0.015,B 0.000,C -180.000} C_DIS
LIN {X -323.818,Y 135.821,Z -44.500,A 0.015,B 0.000,C 180.000} C_DIS
CIRC {X -322.720,Y 132.022,Z -44.500,A 0.015,B 0.000,C 180.000},{X -319.765,Y 129.395,Z -44.500,A 0.015,B 0.000,C -180.000} C_DIS
CIRC {X -307.938,Y 122.709,Z -44.500,A 0.015,B 0.000,C 180.000},{X -297.148,Y 114.453,Z -44.500,A 0.015,B 0.000,C 180.000} C_DIS
CIRC {X -287.430,Y 104.981,Z -44.500,A 0.015,B -0.000,C -180.000},{X -278.711,Y 94.582,Z -44.500,A 0.015,B 0.000,C 180.000} C_DIS
CIRC {X -275.685,Y 90.311,Z -44.500,A 0.015,B 0.000,C -180.000},{X -272.930,Y 85.858,Z -44.500,A 0.015,B 0.000,C 180.000} C_DIS
LIN {X -254.500,Y 52.759,Z -44.500,A 0.015,B 0.000,C 180.000} C_DIS
CIRC {X -251.615,Y 49.788,Z -44.500,A 0.015,B 0.000,C 180.000},{X -247.620,Y 48.697,Z -44.500,A 0.015,B 0.000,C 180.000} C_DIS
LIN {X -145.875,Y 48.697,Z -44.500,A 0.015,B 0.000,C -180.000} C_DIS
CIRC {X -141.898,Y 49.789,Z -44.500,A 0.015,B 0.000,C -180.000},{X -139.036,Y 52.757,Z -44.500,A 0.015,B 0.000,C 180.000} C_DIS
LIN {X -120.092,Y 86.145,Z -44.500,A 0.015,B -0.000,C 180.000} C_DIS
CIRC {X -109.007,Y 101.891,Z -44.500,A 0.015,B -0.000,C -180.000},{X -95.547,Y 115.661,Z -44.500,A 0.015,B 0.000,C -180.000} C_DIS
CIRC {X -90.489,Y 119.692,Z -44.500,A 0.015,B 0.000,C 180.000},{X -85.100,Y 123.269,Z -44.500,A 0.015,B -0.000,C 180.000} C_DIS
CIRC {X -79.489,Y 126.477,Z -44.500,A 0.015,B -0.000,C -180.000},{X -73.736,Y 129.421,Z -44.500,A 0.015,B 0.000,C 180.000} C_DIS
CIRC {X -70.787,Y 132.061,Z -44.500,A 0.015,B -0.000,C -180.000},{X -69.692,Y 135.864,Z -44.500,A 0.015,B 0.000,C -180.000} C_DIS
LIN {X -69.696,Y 256.242,Z -44.500,A 0.015,B 0.000,C 180.000} C_DIS
CIRC {X -72.005,Y 259.030,Z -44.500,A 0.015,B 0.000,C -180.000},{X -75.175,Y 257.282,Z -44.500,A 0.015,B 0.000,C -180.000} C_DIS
CIRC {X -84.923,Y 238.263,Z -44.500,A 0.015,B -0.000,C -180.000},{X -98.203,Y 221.520,Z -44.500,A 0.015,B 0.000,C 180.000} C_DIS
CIRC {X -114.379,Y 207.579,Z -44.500,A 0.015,B 0.000,C 180.000},{X -132.800,Y 196.777,Z -44.500,A 0.015,B 0.000,C 180.000} C_DIS
CIRC {X -152.551,Y 189.901,Z -44.500,A 0.015,B 0.000,C -180.000},{X -173.300,Y 187.286,Z -44.500,A 0.015,B 0.000,C 180.000} C_DIS
LIN {X -214.895,Y 186.858,Z -44.500,A 0.015,B 0.000,C -180.000} C_DIS
CIRC {X -242.578,Y 190.360,Z -44.500,A 0.015,B 0.000,C -180.000},{X -268.518,Y 200.644,Z -44.500,A 0.015,B 0.000,C 180.000} C_DIS

; Continue running program as cascaded execution
Machining2()

END
